{attribute addProperty BoxType "EL6001-0000-0017"}
{attribute addProperty Id "CtrlAT %Q*Ctrl_BE606B1B1621Data_OutAT %Q*ARRAY[0 ..21] OF USINT176220"}
{attribute addProperty CRC "2979260577"}
{attribute addProperty SizeInBites "192"}
{attribute addProperty SizeInBytes "24"}
TYPE COM_Outputs_AC29F8FC :
STRUCT
	{attribute addProperty Name "Ctrl"}
	Ctrl AT %Q* : Ctrl_BE606B1B;
	{attribute addProperty Name "Data_Out"}
	Data_Out AT %Q* : ARRAY[0 ..21] OF USINT;
END_STRUCT
END_TYPE

(* stored: Version 1.2.0.0, ProductVersion 3.1.4024.9
   DUT COM_Outputs_AC29F8FC: Id {7c5a9ae5-8020-4de8-948f-7359ad648d3f} *)
